PROGRAM prgSmartMeter
VAR
//	fbSmartMeter	: FB_KL6781_MBus_Master;	
	int_LiveCount		: INT;	//{#lynus.ag#()}
END_VAR

// fbSmartMeter(eBaudrateMBus := 9600);
logic ();
int_LiveCount:=int_LiveCount+1;

END_PROGRAM

(* stored: Version 1.1.0.1, ProductVersion 3.1.4024.11
   POU prgSmartMeter: Id {c9c25a81-16a4-48e9-8568-6d2b8c776c23}, SpecialFunc None *)
